Fanuc KAREL source: kb00065.KL

-- PROVISIONAL review KL for V770-1; original PC SHA256 f3a39013e6182c3b27dc4ee40e923e637dfd4bd2af1c6a7ca73cac1d1791706e
-- Incomplete behavior may be omitted. Consult companion uncertainty JSON. Do not deploy.
PROGRAM KB00065
%NOLOCKGROUP
BEGIN
  -- UNRESOLVED_PC offsets 5-14; opcodes 3F,75
  -- UNRESOLVED_PC offsets 19-26; opcodes 9D,23
  -- UNRESOLVED_PC offsets 31-38; opcodes 9D,23
  -- UNRESOLVED_PC offsets 43-52; opcodes 3F,75
  -- UNRESOLVED_PC offsets 57-66; opcodes 3F,75
  -- UNRESOLVED_PC offsets 71-78; opcodes 9D,23
  -- UNRESOLVED_PC offsets 83-90; opcodes 9D,23
  -- UNRESOLVED_PC offsets 95-102; opcodes 9D,23
  -- UNRESOLVED_PC offsets 107-165; opcodes 27,22,2A,22,22,22,2A,22,2A,22,22,22,31
  -- UNRESOLVED_PC offsets 170-174; opcodes 7F
END KB00065
